{attribute 'GeneratedUsingTerminal: CU1561--0000'}
{attribute addProperty BoxType "CU1561--0000"}
{attribute addProperty Id "InfoDataAT %I*InfoData_6F19DB2B2"}
{attribute addProperty CRC "532711307"}
{attribute addProperty Size "2"}
TYPE CU1561_1FC0878B :
STRUCT
	{attribute addProperty Name "InfoData"}
	InfoData : InfoData_6F19DB2B;
END_STRUCT
END_TYPE

(* stored: Version 1.2.0.0, ProductVersion 3.1.4024.9
   DUT CU1561_1FC0878B: Id {307e8384-605a-422a-bff5-2fbbc17b95c0} *)
